Staubli VAL3: Control_YesNo.pgx

public program Control_YesNo(string x_sMess (dimensions=1), bool& x_bRes (dimensions=1))
  local num l_nKey
begin
  // title("示教工具头")
  cls()

  gotoxy(3,3)
  put("┌───────────────────────────────┐")
  gotoxy(3,4)
  put("│                               │")
  gotoxy(3,5)
  put("│                               │")
  gotoxy(3,6)
  put("│                               │")
  gotoxy(3,7)
  put("│                               │")
  gotoxy(3,8)
  put("└───────────────────────────────┘")


  gotoxy(12,6)
  put(x_sMess)


  gotoxy(0,13)
  put(right("                                               否  是 ",37))









  while true

    l_nKey=getKey()

    switch l_nKey

      case 277
        x_bRes=false
        return
      break


      case 278
        x_bRes=true
        return
      break


    endSwitch


    delay(0)
  endWhile







end
